FUNCTION_BLOCK CM_Motor IMPLEMENTS  ITF_Motor
VAR
	fb_mem : STRUCT_CM_Motor;
END_VAR

(*
$$$$$$$$\                                                                   $$\       $$$$$$$$\                     $$\                                         $$\                     
$$  _____|                                                                  $$ |      $$  _____|                    \__|                                        \__|                    
$$ |   $$$$$$\   $$$$$$\  $$$$$$$\  $$\  $$\  $$\  $$$$$$\   $$$$$$\   $$$$$$$ |      $$ |      $$$$$$$\   $$$$$$\  $$\ $$$$$$$\   $$$$$$\   $$$$$$\   $$$$$$\  $$\ $$$$$$$\   $$$$$$\  
$$$$$\ \____$$\ $$  __$$\ $$  __$$\ $$ | $$ | $$ |$$  __$$\ $$  __$$\ $$  __$$ |      $$$$$\    $$  __$$\ $$  __$$\ $$ |$$  __$$\ $$  __$$\ $$  __$$\ $$  __$$\ $$ |$$  __$$\ $$  __$$\ 
$$  __|$$$$$$$ |$$ |  \__|$$ |  $$ |$$ | $$ | $$ |$$ /  $$ |$$ /  $$ |$$ /  $$ |      $$  __|   $$ |  $$ |$$ /  $$ |$$ |$$ |  $$ |$$$$$$$$ |$$$$$$$$ |$$ |  \__|$$ |$$ |  $$ |$$ /  $$ |
$$ |  $$  __$$ |$$ |      $$ |  $$ |$$ | $$ | $$ |$$ |  $$ |$$ |  $$ |$$ |  $$ |      $$ |      $$ |  $$ |$$ |  $$ |$$ |$$ |  $$ |$$   ____|$$   ____|$$ |      $$ |$$ |  $$ |$$ |  $$ |
$$ |  \$$$$$$$ |$$ |      $$ |  $$ |\$$$$$\$$$$  |\$$$$$$  |\$$$$$$  |\$$$$$$$ |      $$$$$$$$\ $$ |  $$ |\$$$$$$$ |$$ |$$ |  $$ |\$$$$$$$\ \$$$$$$$\ $$ |      $$ |$$ |  $$ |\$$$$$$$ |
\__|   \_______|\__|      \__|  \__| \_____\____/  \______/  \______/  \_______|      \________|\__|  \__| \____$$ |\__|\__|  \__| \_______| \_______|\__|      \__|\__|  \__| \____$$ |
                                                                                                          $$\   $$ |                                                          $$\   $$ |
      			                                                                                          \$$$$$$  |                                                          \$$$$$$  |
                                                                                                           \______/                                                            \______/ 
*)
fb_mem.STS.State := PackML_StateMachine(State			:= fb_mem.STS.State,
										Start           := fb_mem.CS.Start,
										Stop            := fb_mem.CS.Stop,
										Reset           := fb_mem.CS.Reset,
										Abort           := fb_mem.CS.Abort,
										Clear           := fb_mem.CS.Clear,
										UnSuspend       := fb_mem.CS.UnSuspend,
										Suspend         := fb_mem.CS.Suspend,
										UnHold          := fb_mem.CS.UnHold,
										Hold            := fb_mem.CS.Hold,
										Starting_SC     := fb_mem.STS.Starting_SC,
										Execute_SC      := fb_mem.STS.Execute_SC,
										Completing_SC	:= fb_mem.STS.Completing_SC,
										Resetting_SC    := fb_mem.STS.Resetting_SC,
										Holding_SC      := fb_mem.STS.Holding_SC,
										Unholding_SC    := fb_mem.STS.Unholding_SC,
										Suspending_SC   := fb_mem.STS.Suspending_SC,
										Unsuspending_SC := fb_mem.STS.Unsuspending_SC,
										Aborting_SC     := fb_mem.STS.Aborting_SC,
										Clearing_SC     := fb_mem.STS.Clearing_SC,
										Stopping_SC     := fb_mem.STS.Stopping_SC);

//********************************Auto manual logic***********************************
IF fb_mem.CS.Auto OR fb_mem.HMI.Auto THEN
	fb_mem.STS.Auto := TRUE;
	fb_mem.STS.Manueel := FALSE;
END_IF

IF fb_mem.CS.Manueel OR fb_mem.HMI.Manueel THEN
	fb_mem.STS.Auto := FALSE;
	fb_mem.STS.Manueel := TRUE;
END_IF

//********************************Toerental***********************************

fb_mem.STS.Toerental := fb_mem.CS.Toerental;

//********************************Exeptionhandling***********************************

//********************************Action case***********************************
CASE fb_mem.STS.State OF
	E_State_PackML.IDLE 			:
		//Do nothing
	E_State_PackML.STARTING 		:
		fb_mem.STS.Starting_SC 		:= TRUE;
	E_State_PackML.EXECUTE 			: 
		//Do nothing
	E_State_PackML.COMPLETING		:
		fb_mem.STS.Completing_SC := TRUE;
	E_State_PackML.COMPLETE 		:
		IF fb_mem.CS.Clear AND fb_mem.STS.Auto OR fb_mem.HMI.Clear AND fb_mem.STS.Manueel THEN
			fb_mem.STS.Completing_SC := TRUE;
		END_IF
	E_State_PackML.RESETTING 		:
		FB_init(0,0);
		fb_mem.STS.Resetting_SC 	:= TRUE;
	E_State_PackML.HOLDING 			:
		fb_mem.STS.Unholding_SC		:= TRUE;
	E_State_PackML.HELD 			:
		//Do nothing
	E_State_PackML.UNHOLDING 		:
		fb_mem.STS.Unholding_SC		:= TRUE;
	E_State_PackML.SUSPENDING 		:
		fb_mem.STS.Suspending_SC 	:= TRUE;
	E_State_PackML.SUSPENDED 		:
		fb_mem.CS.Unsuspend 		:= TRUE;
	E_State_PackML.UNSUSPENDING 	:
		fb_mem.STS.Unsuspending_SC 	:= TRUE;
	E_State_PackML.ABORTED			:
		//Do nothing
	E_State_PackML.ABORTING			:
		fb_mem.STS.Aborting_SC 		:= TRUE;
	E_State_PackML.CLEARING 		:
		fb_mem.STS.Clearing_SC 		:= TRUE;
	E_State_PackML.STOPPING 		:
		fb_mem.STS.Stopping_SC 		:= TRUE;
	E_State_PackML.STOPPED 			:
		//Do nothing
		
END_CASE




//Zero all CS signals
fb_mem.CS.Auto			:= FALSE;
fb_mem.CS.Manueel 		:= FALSE;
fb_mem.CS.Abort			:= FALSE;
fb_mem.CS.Reset			:= FALSE;
fb_mem.CS.Richting_L	:= FALSE;
fb_mem.CS.Richting_R	:= FALSE;
fb_mem.CS.Start			:= FALSE;
fb_mem.CS.Stop			:= FALSE;

//Zero all HMI signals
fb_mem.HMI.Auto			:= FALSE;
fb_mem.HMI.Manueel 		:= FALSE;
fb_mem.HMI.Abort		:= FALSE;
fb_mem.HMI.Reset		:= FALSE;
fb_mem.HMI.Richting_L	:= FALSE;
fb_mem.HMI.Richting_R	:= FALSE;
fb_mem.HMI.Start		:= FALSE;
fb_mem.HMI.Stop			:= FALSE;

{warning 'add method implementation '}
METHOD Abort : BOOL
fb_mem.CS.Abort := TRUE;

Abort := fb_mem.CS.Abort;
END_METHOD

PROPERTY Auto : BOOl
GET
AUTO := fb_mem.STS.Auto;
END_GET
SET
fb_mem.CS.Auto := AUTO;
END_SET
END_PROPERTY

METHOD Clear : BOOL
VAR_INPUT
END_VAR
fb_mem.CS.Clear := TRUE;

Clear := fb_mem.CS.Abort;
END_METHOD

{warning 'add property implementation'}
PROPERTY Error_State : E_Motor_Error_State
GET
Error_State := fb_mem.STS.Error_State;
END_GET
END_PROPERTY

METHOD FB_init : BOOL
VAR_INPUT
	bInitRetains : BOOL; // if TRUE, the retain variables are initialized (warm start / cold start)
	bInCopyCode : BOOL;  // if TRUE, the instance afterwards gets moved into the copy code (online change)
END_VAR
fb_mem.STS.State := E_State_PackML.IDLE;
END_METHOD

PROPERTY Manueel : BOOl
GET
Manueel := fb_mem.STS.Manueel;
END_GET
SET
fb_mem.CS.Manueel :=  Manueel;
END_SET
END_PROPERTY

{warning 'add method implementation '}
METHOD Reset : BOOL
fb_mem.CS.Reset := TRUE;

Reset := fb_mem.CS.Reset;
END_METHOD

{warning 'add property implementation'}
PROPERTY Richting_L : BOOL
GET
Richting_L := fb_mem.STS.Richting_L;
END_GET
SET
fb_mem.CS.Richting_L := Richting_L;
END_SET
END_PROPERTY

{warning 'add property implementation'}
PROPERTY Richting_R : BOOL
GET
Richting_R := fb_mem.STS.Richting_R;
END_GET
SET
fb_mem.CS.Richting_R := Richting_R;
END_SET
END_PROPERTY

{warning 'add method implementation '}
METHOD Start : BOOL
fb_mem.CS.Start := TRUE;

Start := fb_mem.CS.Start;
END_METHOD

{warning 'add property implementation'}
PROPERTY State : E_Motor_State
GET
END_GET
END_PROPERTY

{warning 'add method implementation '}
METHOD Stop : BOOL
fb_mem.CS.Stop := TRUE;

Stop := fb_mem.CS.Stop;
END_METHOD

PROPERTY Tag : STRING
GET
Tag := fb_mem.STS.Tag;
END_GET
END_PROPERTY

{warning 'add method implementation '}
METHOD Toerental : INT
fb_mem.CS.Toerental := Toerental;

Toerental := fb_mem.STS.Toerental;
END_METHOD

END_FUNCTION_BLOCK

(* stored: Version 1.1.0.1, ProductVersion 3.1.4024.12
   POU CM_Motor: Id {ad18aa34-53f9-43d5-96e4-85da740b0380}, SpecialFunc None
   Folder Methods: Id {e48a4f7d-e56b-428a-aa1b-5b87c7c2d9fa}
   Folder Properties: Id {bc8caceb-6cf9-4970-a7a5-33f216f9ab87}
   Method Abort: Id {bce41efd-d6b0-4d62-89f5-e33ac87557da}
   Property Auto: Id {11ef47cb-7d87-440a-a57d-2cabaca58e35}
   Get Get: Id {6a6dad5a-3122-4156-a7f6-902e7509088d}
   Set Set: Id {816dc6e2-11f2-441f-a7bc-68dcbe2dd7e0}
   Method Clear: Id {0f8eb475-5a60-456a-a3b0-b756a25c73fb}
   Property Error_State: Id {e515215c-6fc9-4b62-8fc6-8b2fbbaf48cb}
   Get Get: Id {f220728e-61e0-4b32-9b95-9b2cd9b4bf16}
   Method FB_init: Id {b57a1db5-23e5-4a22-9fd5-673c65f1eb7c}
   Property Manueel: Id {7c431163-01ea-4de3-ba47-a54ca14c245f}
   Get Get: Id {76c0c133-7dce-466d-af0b-b4f6f0a95c4b}
   Set Set: Id {f1098c66-0c9f-45a5-9d18-b0c13f2df4b6}
   Method Reset: Id {9ebe56cb-ee7c-443c-9b93-4574a33eba76}
   Property Richting_L: Id {acd82104-10c0-4d3d-b202-3582cda0f6aa}
   Get Get: Id {254eef6c-679d-4955-9374-8c48813a2eba}
   Set Set: Id {971f8c41-0eec-4c04-8969-13b6e9bb900e}
   Property Richting_R: Id {1dfa9288-7cf5-4117-bb7a-1871dc8acb27}
   Get Get: Id {c9301737-e65a-4566-b592-b9a0f81a954d}
   Set Set: Id {c093fe9c-b698-4b4c-be3d-d0eea63cb1c9}
   Method Start: Id {d85189c8-d167-4ff9-9393-dd18fc880ed7}
   Property State: Id {b265f892-f5e4-4964-b773-e12474a75895}
   Get Get: Id {d9b17dd7-10ff-4cfa-a319-4423eeaaebb7}
   Method Stop: Id {cf8e2e14-1e28-43cd-9de6-6cddfbbd163d}
   Property Tag: Id {fefd0db7-e012-4728-b2c5-4de1f2c675d0}
   Get Get: Id {46ff3736-98f0-4078-846d-f939f5f220ac}
   Method Toerental: Id {648fbdfc-50d6-45b6-9f05-5bc65d6066b2} *)
